FUNCTION F_CreateDynText : ST_Text
VAR_INPUT
	wsName		: WSTRING;	//standard name
	nNameId		: INT;		//example simatic hmi
END_VAR
VAR
END_VAR

F_CreateDynText.wsName := wsName;
F_CreateDynText.wsNameId := wsName;
F_CreateDynText.nNameId := nNameId;

END_FUNCTION

(* stored: Version 1.1.0.1, ProductVersion 3.1.4024.12
   POU F_CreateDynText: Id {0838a504-6744-476d-bcb9-033faff7e366}, SpecialFunc None *)
